// CODESYS_Control_x86_Arca_Control_SM/Application/TCPIP Control/TCP_Command_Extract_And_Analysis
FUNCTION_BLOCK TCP_Command_Extract_And_Analysis
VAR_INPUT
	InData : STRING;
	InDataSize : CAA.SIZE;
	InData_Valid : BOOL;
	OutRobot_State : Robot_State;
END_VAR
VAR_OUTPUT
	Command_Valid : BOOL;
	Command : robot_command_via_tcp;
	Response : ARRAY [0..255] OF BYTE;
	Response_Data_Size : CAA.SIZE;
	Response_Valid : BOOL;
	Error : BOOL;
	ErrorMassage : STRING;
END_VAR
VAR
	newDataSize : INT;
	i : INT;
	y : INT;
	state : INT := 0;
	charInData : POINTER TO BYTE;
	charStartF : BYTE := 40; // (
	charStartS : BYTE := 41; // )
	charMid : BYTE := 59; // ;
	charEndF : BYTE := 91; // [
	charEndS : BYTE := 93; // ]
	charAU : BYTE := 65;	// A
	charZU : BYTE := 90;	// Z
	charAL : BYTE := 97;	// a
	charZL : BYTE := 122;	// z
	charMinus : BYTE := 45; // -
	charPeriod : BYTE := 46; // .
	char0 : BYTE := 48; // 0
	char9 : BYTE := 57; // 9
	cache : ARRAY [0..10] OF BYTE;
	cacheCleaner : ARRAY [0..10] OF BYTE;
	
	tag : STRING;
	tagPointer : POINTER TO STRING;
	tagPass : STRING(12);
	
	content : STRING;
	contentPointer : POINTER TO STRING;
	contentNum : REAL;
	_defult_cmd : robot_command_via_tcp;
	
	
	// out going data process
	old_robot_state : Robot_State;
	old_gesture_state : ARRAY [0..8] OF BYTE := [40, 71, 101, 115, 116, 41, 48, 48, 59]; //(Gest)00;
	old_Grab_state : ARRAY [0..7] OF BYTE := [40, 71, 114, 97, 98, 41, 48, 59]; //(Grab)0;
	old_Hand_Enb_state : ARRAY [0..7] OF BYTE := [40, 72, 69, 110, 98, 41, 48, 59]; //(HEnb)0;
	old_Hand_Enb_Err_state : ARRAY [0..10] OF BYTE := [40, 72, 69, 110, 98, 69, 114, 114, 41, 48, 59]; //(HEnbErr)0;
	old_Hand_Mov_Err_state : ARRAY [0..10] OF BYTE := [40, 72, 77, 111, 118, 69, 114, 114, 41, 48, 59]; //(HMovErr)0;
	old_Robot_Mov_Err_state : ARRAY [0..10] OF BYTE := [40, 82, 77, 111, 118, 69, 114, 114, 41, 48, 59]; //(RMovErr)0;
	old_CNC_Executing_state : ARRAY [0..9] OF BYTE := [40, 67, 78, 67, 105, 110, 103, 41, 48, 59]; //(CNCing)0;
	old_CNC_Err_state : ARRAY [0..9] OF BYTE := [40, 67, 78, 67, 69, 72, 72, 41, 48, 59]; //(CNCErr)0;
	old_CNC_Done_state : ARRAY [0..10] OF BYTE := [40, 67, 78, 67, 68, 111, 110, 110, 41, 48, 59]; //(CNCDone)0;
	
	data_end : ARRAY [0..1] OF BYTE := [13, 10];
	og_i : INT;
	og_num_counter : INT;
	
	abc : INT;
	message_sending_timer : ton;
END_VAR

IF Command_Valid THEN
	command_Valid := FALSE; // reset flag after one cycle
	Command := _defult_cmd;	// all content value will only save for one cycle
END_IF;

// process income data
IF (INData_valid AND InDataSize > 0) THEN
	charInData := ADR(InData);
	newDataSize := UDINT_TO_INT(InDataSize);
	Error := FALSE;
	i := 0;
	WHILE i < newDataSize DO
		CASE state OF
			-9:
				IF charInData^ = 93 THEN
					Command_Valid := TRUE;
					i := i + 1;
					state := 0; // if read ]
				ELSE state := 999;
				END_IF
			-8:
				IF charInData^ = 10 THEN
					charInData := charInData + 1;
					i := i + 1;
					state := -9; // if read LF
				ELSE state := 999;
				END_IF
			-7:
				IF charInData^ = 91 THEN
					charInData := charInData + 1;
					i := i + 1;
					state := -8; // if read [
				ELSE state := 999;
				END_IF
			-6:
				IF charInData^ = 93 THEN
					charInData := charInData + 1;
					i := i + 1;
					state := -7; // if read ]
				ELSE state := 999;
				END_IF
			-5:
				IF charInData^ = 13 THEN
					charInData := charInData + 1;
					i := i + 1;
					state := -6; // if read CR
				ELSE state := 999;
				END_IF
			0:
				IF (charInData^ = charStartF) THEN // if read (
					charInData := charInData + 1;
					i := i + 1;
					y := 0;
					state := 10;
				ELSIF charInData^ = charEndF THEN // if read [
					charInData := charInData + 1;
					i := i + 1;
					state := -5;
				ELSE state := 999;
				END_IF
			10:	// exturct laybel
				// if is not ) and not reach end of text and no error
				WHILE (charInData^ <> charStartS) AND (i < newDataSize) AND state = 10 DO
					// if is reading english letter
					IF (CharInData^ >= charAU AND CharInData^ <= charZU) OR (CharInData^ >= charAL AND CharInData^ <= charZL) THEN	
						cache[y] := CharInData^;
						y := y + 1;
						i := i + 1;
						IF i < newDataSize THEN	// only move pointer futher if is not reach the end of text
							charInData := charInData + 1;
						END_IF
					ELSE state := 999;
					END_IF
				END_WHILE
				IF charInData^ = charStartS AND i < newDataSize THEN	// if is ) and not reach end of text
					charInData := charInData + 1;
					i := i + 1;
					y := 0;
					tagPointer := ADR(cache);
					tag := tagPointer^;
					cache := cacheCleaner;
					state := 20;
				END_IF
			20:	// extruct data
				// if is not ; and not reach end of text and no error
				WHILE (charInData^ <> charMid) AND (i < newDataSize) AND state = 20 DO
					// if is reading numbers and - and .
					IF (CharInData^ >= charMinus AND CharInData^ <= charPeriod) OR (CharInData^ >= char0 AND CharInData^ <= char9) THEN
						cache[y] := CharInData^;
						y := y + 1;
						i := i + 1;
						IF i < newDataSize THEN	// only move pointer futher if is not reach the end of text
							charInData := charInData + 1;
						END_IF
					ELSE state := 999;
					END_IF
				END_WHILE
				IF charInData^ = charMid AND i < newDataSize THEN	// if is ; and not reach end of text
					charInData := charInData + 1;
					i := i + 1;
					y := 0;
					contentPointer := ADR(cache);
					content := contentPointer^;
					cache := cacheCleaner;
					contentNum := STRING_TO_REAL(content);
					state := 30;
				END_IF
			30:	// asign data, new label add here
				IF tag = 'X' THEN
					Command.X_Axis_Valid := TRUE;
					Command.X_value := contentNum;
				ELSIF tag = 'Y' THEN
					Command.Y_Axis_Valid := TRUE;
					Command.Y_value := contentNum;
				ELSIF tag = 'Z' THEN
					Command.Z_Axis_Valid := TRUE;
					Command.Z_value := contentNum;
				ELSIF tag = 'GRAB' THEN
					Command.Grab_Valid := TRUE;
					IF contentNum = 1 THEN
						Command.Grab_state := TRUE;
					ELSE 
						Command.Grab_state := FALSE;
					END_IF
				ELSIF tag = 'GEST' THEN
					Command.Gesture_Valid := TRUE;
					CASE (REAL_TO_INT(contentnum)) OF
						0:
							Command.Gesture_Num := 0;
						1:
							Command.Gesture_Num := 1;
						2:
							Command.Gesture_Num := 2;
						3:
							Command.Gesture_Num := 3;
						4:
							Command.Gesture_Num := 4;
						5:
							Command.Gesture_Num := 5;
						6:
							Command.Gesture_Num := 6;
						10:
							Command.Gesture_Num := 10;
						11:
							Command.Gesture_Num := 11;
						12:
							Command.Gesture_Num := 12;
						13:
							Command.Gesture_Num := 13;
						14:
							Command.Gesture_Num := 14;
						15:
							Command.Gesture_Num := 15;
						16:
							Command.Gesture_Num := 16;
						17:
							Command.Gesture_Num := 17;
					END_CASE
					
				ELSIF tag = 'HENB' THEN	// hand enable
					Command.Enabl_Hand_Valid := TRUE;
					IF contentNum = 1 THEN
						Command.Enabl_Hand_state := TRUE;
					ELSE 
						Command.Enabl_Hand_state := FALSE;
					END_IF
				ELSIF tag = 'HDem' THEN	// hand demo
					Command.Gesture_Demo_Valid := TRUE;
					IF contentNum = 1 THEN
						Command.Gesture_Demo_state := TRUE;
					ELSE 
						Command.Gesture_Demo_state := FALSE;
					END_IF
				ELSIF tag = 'CNC' THEN	// CNC program move command
					Command.CNC_Mov_Valid := TRUE;
					Command.CNC_Mov_Program_Num := REAL_TO_INT(contentnum);
				END_IF
				state := 0;
			999:
				i := newDataSize;
				state := 0;
				Error := TRUE;
				ErrorMassage := 'Error Data not match rule';
		END_CASE
	END_WHILE
END_IF

Response_Valid := FALSE;
message_sending_timer(in := TRUE, pt := T#100MS);
// process outgoing data
IF
	(
	outrobot_state.Gesture_State <> old_robot_state.Gesture_State
	OR outrobot_state.Grab_State <> old_robot_state.Grab_State
	OR outrobot_state.Hand_Enabled <> old_robot_state.Hand_Enabled
	OR outrobot_state.Hand_Enb_Err <> old_robot_state.Hand_Enb_Err
	OR outrobot_state.Hand_Mov_Err <> old_robot_state.Hand_Mov_Err
	OR outrobot_state.Robot_Mov_Err <> old_robot_state.Robot_Mov_Err
	)
	AND
	message_sending_timer.Q
THEN
	message_sending_timer(in := FALSE);
	abc := abc +1;
	//debug:= TRUE;
	og_num_counter := 0;
	
	// gesture state
	IF outrobot_state.Gesture_State <> old_robot_state.Gesture_State THEN
			
		CASE outrobot_state.Gesture_State OF
			0:
				old_gesture_state[6] := 48;
				old_gesture_state[7] := 48;
			1:
				old_gesture_state[6] := 48;
				old_gesture_state[7] := 49;
			2:
				old_gesture_state[6] := 48;
				old_gesture_state[7] := 50;
			3:
				old_gesture_state[6] := 48;
				old_gesture_state[7] := 51;
			4:
				old_gesture_state[6] := 48;
				old_gesture_state[7] := 52;
			5:
				old_gesture_state[6] := 48;
				old_gesture_state[7] := 53;
			6:
				old_gesture_state[6] := 48;
				old_gesture_state[7] := 54;
			10:
				old_gesture_state[6] := 49;
				old_gesture_state[7] := 48;
			11:
				old_gesture_state[6] := 49;
				old_gesture_state[7] := 49;
			12:
				old_gesture_state[6] := 49;
				old_gesture_state[7] := 50;
			13:
				old_gesture_state[6] := 49;
				old_gesture_state[7] := 51;
			14:
				old_gesture_state[6] := 49;
				old_gesture_state[7] := 52;
			15:
				old_gesture_state[6] := 49;
				old_gesture_state[7] := 53;
			16:
				old_gesture_state[6] := 49;
				old_gesture_state[7] := 54;
			17:
				old_gesture_state[6] := 49;
				old_gesture_state[7] := 55;
		END_CASE
		
		FOR og_i := 0 TO UDINT_TO_INT(SIZEOF(old_gesture_state)) - 1 DO
			Response[og_num_counter] := old_gesture_state[og_i];
			og_num_counter := og_num_counter + 1;
		END_FOR
	END_IF
	
	// Grab state
	IF outrobot_state.Grab_State <> old_robot_state.Grab_State THEN
		IF outrobot_state.Grab_State THEN	// if true
			old_Grab_state[6] := 49;
		ELSE
			old_Grab_state[6] := 48;
		END_IF
		
		FOR og_i := 0 TO UDINT_TO_INT(SIZEOF(old_Grab_state)) - 1 DO
			Response[og_num_counter] := old_Grab_state[og_i];
			og_num_counter := og_num_counter + 1;
		END_FOR
	END_IF
	
	// hand enable state
	IF outrobot_state.Hand_Enabled <> old_robot_state.Hand_Enabled THEN
		IF outrobot_state.Hand_Enabled THEN	// if true
			old_Hand_Enb_state[6] := 49;
		ELSE
			old_Hand_Enb_state[6] := 48;
		END_IF
		
		FOR og_i := 0 TO UDINT_TO_INT(SIZEOF(old_Hand_Enb_state)) - 1 DO
			Response[og_num_counter] := old_Hand_Enb_state[og_i];
			og_num_counter := og_num_counter + 1;
		END_FOR
	END_IF
	
	// Hand enable error state
	IF outrobot_state.Hand_Enb_Err <> old_robot_state.Hand_Enb_Err THEN
		IF outrobot_state.Hand_Enb_Err THEN	// if true
			old_Hand_Enb_Err_state[9] := 49;
		ELSE
			old_Hand_Enb_Err_state[9] := 48;
		END_IF
		
		FOR og_i := 0 TO UDINT_TO_INT(SIZEOF(old_Hand_Enb_Err_state)) - 1 DO
			Response[og_num_counter] := old_Hand_Enb_Err_state[og_i];
			og_num_counter := og_num_counter + 1;
		END_FOR
	END_IF
	
	// hand move error state
	IF outrobot_state.Hand_Mov_Err <> old_robot_state.Hand_Mov_Err THEN
		IF outrobot_state.Hand_Mov_Err THEN	// if true
			old_Hand_Mov_Err_state[9] := 49;
		ELSE
			old_Hand_Mov_Err_state[9] := 48;
		END_IF
		
		FOR og_i := 0 TO UDINT_TO_INT(SIZEOF(old_Hand_Mov_Err_state)) - 1 DO
			Response[og_num_counter] := old_Hand_Mov_Err_state[og_i];
			og_num_counter := og_num_counter + 1;
		END_FOR
	END_IF
	
	// robot move error state
	IF outrobot_state.Robot_Mov_Err <> old_robot_state.Robot_Mov_Err THEN
		IF outrobot_state.Robot_Mov_Err THEN	// if true
			old_Robot_Mov_Err_state[9] := 49;
		ELSE
			old_Robot_Mov_Err_state[9] := 48;
		END_IF
		
		FOR og_i := 0 TO UDINT_TO_INT(SIZEOF(old_Robot_Mov_Err_state)) - 1 DO
			Response[og_num_counter] := old_Robot_Mov_Err_state[og_i];
			og_num_counter := og_num_counter + 1;
		END_FOR
	END_IF
	
	// CNC executing or not
	IF outrobot_state.CNC_Executing <> old_robot_state.CNC_Executing THEN
		IF outrobot_state.CNC_Executing THEN	// if true
			old_CNC_Executing_state[8] := 49;
		ELSE
			old_CNC_Executing_state[8] := 48;
		END_IF
		
		FOR og_i := 0 TO UDINT_TO_INT(SIZEOF(old_CNC_Executing_state)) - 1 DO
			Response[og_num_counter] := old_CNC_Executing_state[og_i];
			og_num_counter := og_num_counter + 1;
		END_FOR
	END_IF
	
	// CNC Error
	IF outrobot_state.CNC_Execute_Err <> old_robot_state.CNC_Execute_Err THEN
		IF outrobot_state.CNC_Execute_Err THEN	// if true
			old_CNC_Err_state[8] := 49;
		ELSE
			old_CNC_Err_state[8] := 48;
		END_IF
		
		FOR og_i := 0 TO UDINT_TO_INT(SIZEOF(old_CNC_Err_state)) - 1 DO
			Response[og_num_counter] := old_CNC_Err_state[og_i];
			og_num_counter := og_num_counter + 1;
		END_FOR
	END_IF
	
	// CNC finish or not
	IF outrobot_state.CNC_Execute_Done <> old_robot_state.CNC_Execute_Done THEN
		IF outrobot_state.CNC_Execute_Done THEN	// if true
			old_CNC_Done_state[9] := 49;
		ELSE
			old_CNC_Done_state[9] := 48;
		END_IF
		
		FOR og_i := 0 TO UDINT_TO_INT(SIZEOF(old_CNC_Done_state)) - 1 DO
			Response[og_num_counter] := old_CNC_Done_state[og_i];
			og_num_counter := og_num_counter + 1;
		END_FOR
	END_IF
	
	(*	templet for new laybel
	// CNC executing or not
	IF outrobot_state. <> old_robot_state. THEN
		IF outrobot_state. THEN	// if true
			[6] := 49;
		ELSE
			[6] := 48;
		END_IF
		
		FOR og_i := 0 TO UDINT_TO_INT(SIZEOF()) - 1 DO
			Response[og_num_counter] := [og_i];
			og_num_counter := og_num_counter + 1;
		END_FOR
	END_IF
	*)
	
	// add ending
	FOR og_i := 0 TO 1 DO
		Response[og_num_counter] := 91;	// [
		og_num_counter := og_num_counter + 1;
		Response[og_num_counter] := data_end[og_i];	// CR, LF
		og_num_counter := og_num_counter + 1;
		Response[og_num_counter] := 93;	// ]
		og_num_counter := og_num_counter + 1;
	END_FOR
	
	Response_Data_Size := INT_TO_UDINT(og_num_counter);
	Response_Valid := TRUE;
	old_robot_state := outrobot_state;
END_IF

END_FUNCTION_BLOCK

// CODESYS_Control_x86_Arca_Control_SM/Application/Testment_Cartesian_Laser_Platform_Test/Cartesian_Laser_Circle_Testment
PROGRAM Cartesian_Laser_Circle_Testment	// draw circle as quick as possible
VAR
	
	EnableRobot : BOOL;
	
	enb_axis_and_robot : AuxAxis_PowerOn;
	circle_State : INT;
	col_begain : ARRAY [1..6] OF REAL := [0,0,0,0,0,0];
	row_begain : ARRAY [1..6] OF REAL := [0,0,0,0,0,0];
	col_num_total: BYTE := 10;
	row_num_total : BYTE := 10;
END_VAR


enb_axis_and_robot(enable := EnableRobot);

if not enablerobot then
	circle_State := 0;
END_IF
CASE circle_State OF
	0:
		IF enb_axis_and_robot.Done THEN
			circle_State := 10;
		END_IF
	10:
	
END_CASE

END_PROGRAM
